Omron CX-Programmer project NewProject (CX-Programmer 9.61)

# PLC UAS_Fix: CP1E N20

## Global symbols (name address type ; comment)
0.00 BOOL  ; Start
0.01 BOOL  ; Stop
0.02 BOOL  ; Sensor Level Minimum
0.03 BOOL  ; Sensor Maksimum
0.04 BOOL  ; Sensor Minimum
0.05 BOOL  ; Sensor Minimum
100.00 BOOL  ; Valve Penguras
100.01 BOOL  ; Valve Air Bersih
100.02 BOOL  ; Valve Air Limbah
100.03 BOOL  ; Sensor Maksimal
100.04 BOOL  ; Mixer Motor
100.05 BOOL  ; Pompa Klorin
100.06 BOOL  ; Blower 1
100.07 BOOL  ; Blower 2
100.08 BOOL  ; Pompa Keluar
T000 BOOL  ; Timer Valve 1
T001 BOOL  ; Timer Valve 2
T002 BOOL  ; Timer Mixer
T003 BOOL  ; Timer Blower 1
T004 BOOL  ; Timer Blower 2
W0.00 BOOL  ; Coil 1
W0.01 BOOL  ; Keep 1
W0.02 BOOL  ; Coil 2
W0.03 BOOL  ; Keep 2

## Program NewProgram1 (cyclic task 0)

### Section Section1

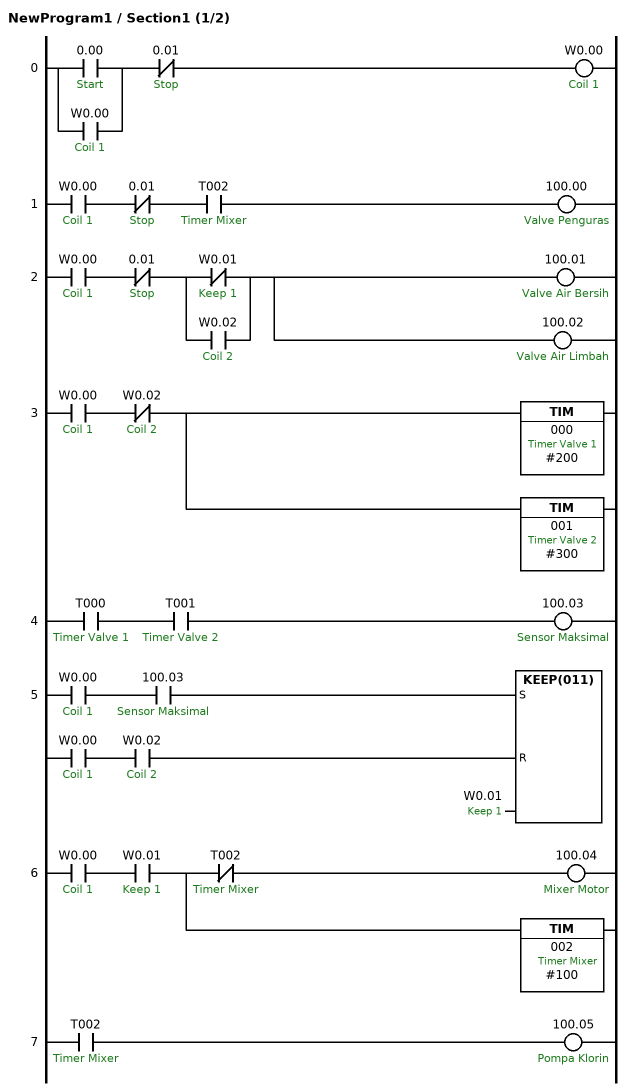
; rung 0
LD 0.00  ; Start
OR W0.00  ; Coil 1
ANDNOT 0.01  ; Stop
OUT W0.00  ; Coil 1
; rung 1
LD W0.00  ; Coil 1
ANDNOT 0.01  ; Stop
AND T002  ; Timer Mixer
OUT 100.00  ; Valve Penguras
; rung 2
LD W0.00  ; Coil 1
ANDNOT 0.01  ; Stop
LDNOT W0.01  ; Keep 1
OR W0.02  ; Coil 2
ANDLD
OUT 100.01  ; Valve Air Bersih
OUT 100.02  ; Valve Air Limbah
; rung 3
LD W0.00  ; Coil 1
ANDNOT W0.02  ; Coil 2
TIM 000 #200  ; Timer Valve 1
TIM 001 #300  ; Timer Valve 2
; rung 4
LD T000  ; Timer Valve 1
AND T001  ; Timer Valve 2
OUT 100.03  ; Sensor Maksimal
; rung 5
LD W0.00  ; Coil 1
AND 100.03  ; Sensor Maksimal
LD W0.00  ; Coil 1
AND W0.02  ; Coil 2
KEEP(011) W0.01  ; Keep 1
; rung 6
LD W0.00  ; Coil 1
AND W0.01  ; Keep 1
OUT TR0
ANDNOT T002  ; Timer Mixer
OUT 100.04  ; Mixer Motor
LD TR0
TIM 002 #100  ; Timer Mixer
; rung 7
LD T002  ; Timer Mixer
OUT 100.05  ; Pompa Klorin

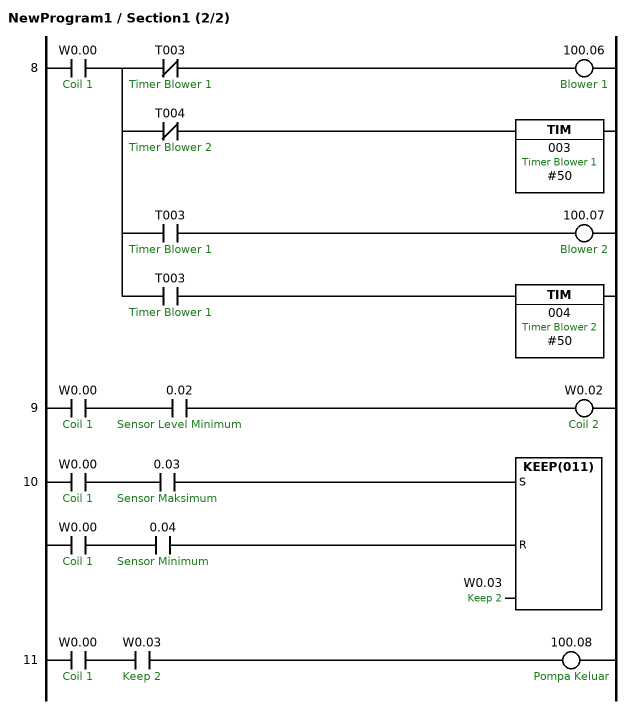
; rung 8
LD W0.00  ; Coil 1
OUT TR0
ANDNOT T003  ; Timer Blower 1
OUT 100.06  ; Blower 1
LD TR0
ANDNOT T004  ; Timer Blower 2
TIM 003 #50  ; Timer Blower 1
LD TR0
AND T003  ; Timer Blower 1
OUT 100.07  ; Blower 2
LD TR0
AND T003  ; Timer Blower 1
TIM 004 #50  ; Timer Blower 2
; rung 9
LD W0.00  ; Coil 1
AND 0.02  ; Sensor Level Minimum
OUT W0.02  ; Coil 2
; rung 10
LD W0.00  ; Coil 1
AND 0.03  ; Sensor Maksimum
LD W0.00  ; Coil 1
AND 0.04  ; Sensor Minimum
KEEP(011) W0.03  ; Keep 2
; rung 11
LD W0.00  ; Coil 1
AND W0.03  ; Keep 2
OUT 100.08  ; Pompa Keluar

### Section END
; rung 0
END(001)